// TIA Portal V17 export
// export: Created 2023-12-22T15:07:59.1760548Z, ExportSetting WithDefaults, DisplayName Totally Integrated Automation Portal, DisplayVersion V17, DisplayName TIA Portal Openness, DisplayVersion V17, DisplayName TIA Portal Version Control Interface, DisplayVersion V17, DisplayName STEP 7 Professional, DisplayVersion V17, DisplayName STEP 7 Safety, DisplayVersion V17, DisplayName WinCC Advanced, DisplayVersion V17
FUNCTION_BLOCK "PS_cnt"   // FB12, LAD
{ S7_Optimized_Access := 'FALSE' }
VERSION : 0.1
// stored: AutoNumber false, IsIECCheckEnabled false, SetENOAutomatically false, UDAEnableTagReadback false
   VAR_INPUT
      SP : Real;
      REQ : Int;
   END_VAR
   VAR_IN_OUT
      cnt : Int;   // Число насосов в работе
   END_VAR
   VAR DB_SPECIFIC
      Select_CMD : Bool;   // Запрос выбора насоса
      Select_Mode : Bool;   // 0 - для останова, 1 - для запуска
      Select_PS : Int;   // Выбранный насос
      PS_Add_Ready : Bool;   // Насосы вышли на общую точку
      PS_Add_CMD : Bool;   // Запрос выхода на общую точку
      SP_Low : Real := 40.0;   // Нижняя рабочая точка
      SP_High { S7_SetPoint := 'True'} : Real := 45.0;   // Верхняя рабочая точка
      SP_Min { S7_SetPoint := 'True'} : Real := 36.0;   // Точка открытия обратного клапана
      cnt_delta { S7_SetPoint := 'True'} : Real := 0.5;   // Смещение точки открытия обратного клапана на 1 работающий насос
      "Step" : Int;
      REQ_cnt : Int;
      PS_R_OFF : Int;   // Насос для отключения при ротации
      PS_R_ON : Int;   // Насос для запуска при ротации
      pos : Array[0..15] of Bool;
      tmp : Array[0..15] of Real;
   END_VAR
   VAR
      T_Delay_ON { S7_SetPoint := 'True'} : "Time_M";   // Задержка запуска след. насоса
      T_Delay_OFF { S7_SetPoint := 'True'} : "Time_M";   // Задержка останова след. насоса
   END_VAR
   VAR_TEMP
      x_delta : Real;
   END_VAR
   VAR_TEMP   // added for the SCL form of the ladder/FBD networks
      _w1 : Bool;
      _w2 : Bool;
      _w3 : Bool;
      _w4 : Bool;
      _w5 : Bool;
      _w6 : Bool;
      _w7 : Bool;
      _w8 : Bool;
   END_VAR
BEGIN

REGION Network 1: Коррекция нижней рабочей точки по числу насосов
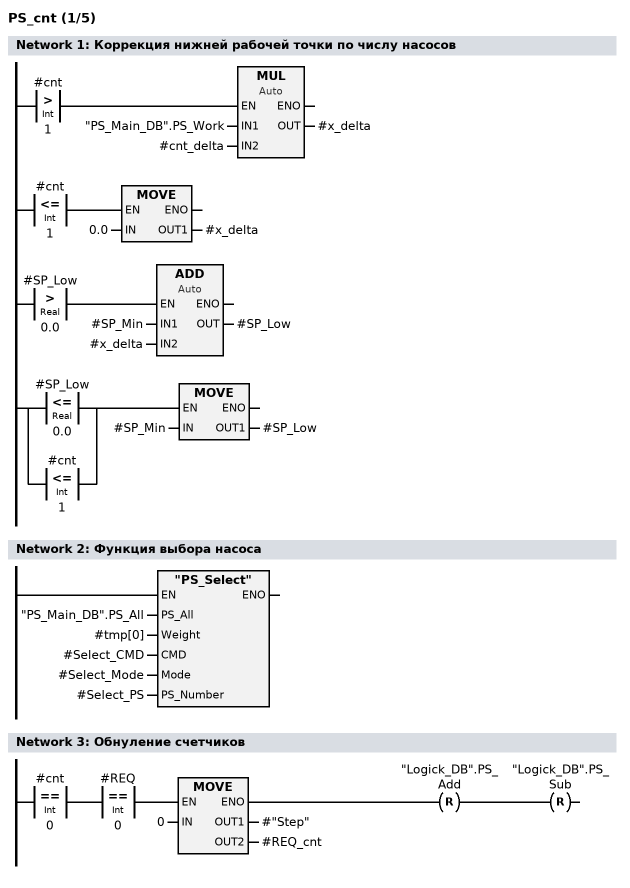
   RUNG wire#powerrail
      { S7_Templates := "SrcType := Int" } GT_Contact(in1 := #cnt, in2 := 1)
      Mul(in1 := "PS_Main_DB".PS_Work, in2 := #cnt_delta, out => #x_delta)
   END_RUNG
   RUNG wire#powerrail
      { S7_Templates := "SrcType := Int" } LE_Contact(in1 := #cnt, in2 := 1)
      Move(in := 0.0, out1 => #x_delta)
   END_RUNG
   RUNG wire#powerrail
      { S7_Templates := "SrcType := Real" } GT_Contact(in1 := #SP_Low, in2 := 0.0)
      Add(in1 := #SP_Min, in2 := #x_delta, out => #SP_Low)
   END_RUNG
   RUNG wire#powerrail
      { S7_Templates := "SrcType := Real" } LE_Contact(in1 := #SP_Low, in2 := 0.0)
      wire#w1
      Move(in := #SP_Min, out1 => #SP_Low)
   END_RUNG
   RUNG wire#powerrail
      { S7_Templates := "SrcType := Int" } LE_Contact(in1 := #cnt, in2 := 1)
   END_RUNG wire#w1
   // the same network as SCL:
   IF #cnt > 1 THEN #x_delta := "PS_Main_DB".PS_Work * #cnt_delta; END_IF;
   IF #cnt <= 1 THEN #x_delta := 0.0; END_IF;
   IF #SP_Low > 0.0 THEN #SP_Low := #SP_Min + #x_delta; END_IF;
   IF (#SP_Low <= 0.0) OR (#cnt <= 1) THEN #SP_Low := #SP_Min; END_IF;
END_REGION

REGION Network 2: Функция выбора насоса
   RUNG wire#powerrail
      "PS_Select"(PS_All := "PS_Main_DB".PS_All, Weight := #tmp[0], CMD := #Select_CMD, Mode := #Select_Mode, PS_Number := #Select_PS)
   END_RUNG
   // the same network as SCL:
   "PS_Select"(PS_All := "PS_Main_DB".PS_All,
               Weight := #tmp[0],
               CMD := #Select_CMD,
               Mode := #Select_Mode,
               PS_Number := #Select_PS);
END_REGION

REGION Network 3: Обнуление счетчиков
   RUNG wire#powerrail
      { S7_Templates := "SrcType := Int" } EQ_Contact(in1 := #cnt, in2 := 0)
      { S7_Templates := "SrcType := Int" } EQ_Contact(in1 := #REQ, in2 := 0)
      Move(in := 0, out1 => #"Step", out2 => #REQ_cnt)
      R_Coil( "Logick_DB".PS_Add )
      R_Coil( "Logick_DB".PS_Sub )
   END_RUNG
   // the same network as SCL:
   IF (#cnt = 0) AND (#REQ = 0) THEN
       #"Step" := 0;
       #REQ_cnt := 0;
       "Logick_DB".PS_Add := FALSE;
       "Logick_DB".PS_Sub := FALSE;
   END_IF;
END_REGION

REGION Network 4: Запуск первого насоса
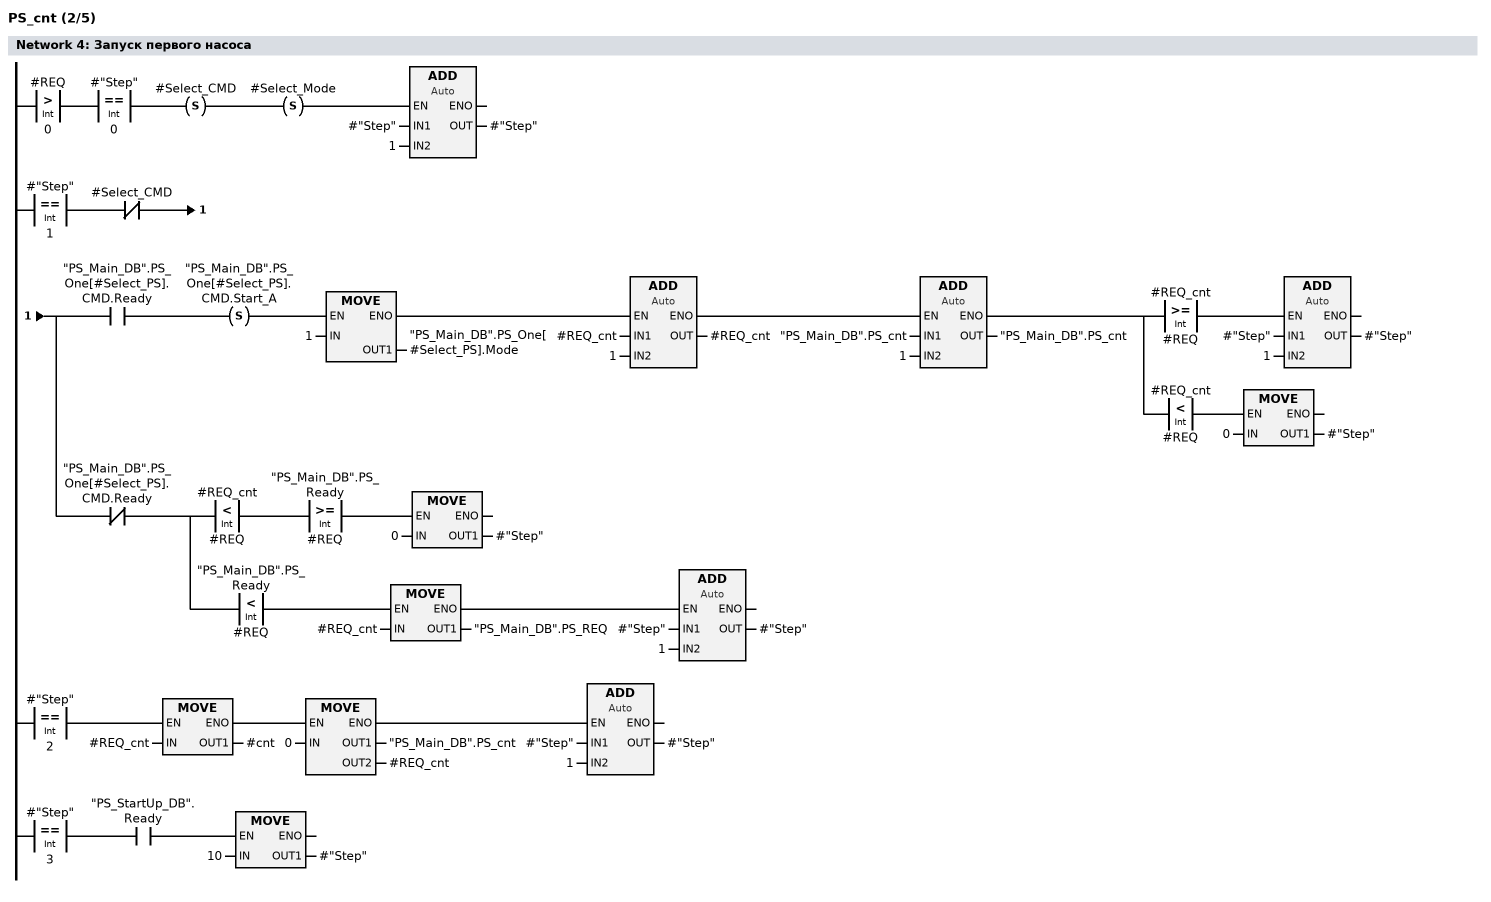
   RUNG wire#powerrail
      { S7_Templates := "SrcType := Int" } GT_Contact(in1 := #REQ, in2 := 0)
      { S7_Templates := "SrcType := Int" } EQ_Contact(in1 := #"Step", in2 := 0)
      S_Coil( #Select_CMD )
      S_Coil( #Select_Mode )
      Add(in1 := #"Step", in2 := 1, out => #"Step")
   END_RUNG
   RUNG wire#powerrail
      { S7_Templates := "SrcType := Int" } EQ_Contact(in1 := #"Step", in2 := 1)
      I_Contact( #Select_CMD )
      wire#w1
      Contact( "PS_Main_DB".PS_One[#Select_PS].CMD.Ready )
      S_Coil( "PS_Main_DB".PS_One[#Select_PS].CMD.Start_A )
      Move(in := 1, out1 => "PS_Main_DB".PS_One[#Select_PS].Mode)
      Add(in1 := #REQ_cnt, in2 := 1, out => #REQ_cnt)
      Add(in1 := "PS_Main_DB".PS_cnt, in2 := 1, out => "PS_Main_DB".PS_cnt)
      wire#w2
      { S7_Templates := "SrcType := Int" } GE_Contact(in1 := #REQ_cnt, in2 := #REQ)
      Add(in1 := #"Step", in2 := 1, out => #"Step")
   END_RUNG
   RUNG wire#w2
      { S7_Templates := "SrcType := Int" } LT_Contact(in1 := #REQ_cnt, in2 := #REQ)
      Move(in := 0, out1 => #"Step")
   END_RUNG
   RUNG wire#w1
      I_Contact( "PS_Main_DB".PS_One[#Select_PS].CMD.Ready )
      wire#w3
      { S7_Templates := "SrcType := Int" } LT_Contact(in1 := #REQ_cnt, in2 := #REQ)
      { S7_Templates := "SrcType := Int" } GE_Contact(in1 := "PS_Main_DB".PS_Ready, in2 := #REQ)
      Move(in := 0, out1 => #"Step")
   END_RUNG
   RUNG wire#w3
      { S7_Templates := "SrcType := Int" } LT_Contact(in1 := "PS_Main_DB".PS_Ready, in2 := #REQ)
      Move(in := #REQ_cnt, out1 => "PS_Main_DB".PS_REQ)
      Add(in1 := #"Step", in2 := 1, out => #"Step")
   END_RUNG
   RUNG wire#powerrail
      { S7_Templates := "SrcType := Int" } EQ_Contact(in1 := #"Step", in2 := 2)
      Move(in := #REQ_cnt, out1 => #cnt)
      Move(in := 0, out1 => "PS_Main_DB".PS_cnt, out2 => #REQ_cnt)
      Add(in1 := #"Step", in2 := 1, out => #"Step")
   END_RUNG
   RUNG wire#powerrail
      { S7_Templates := "SrcType := Int" } EQ_Contact(in1 := #"Step", in2 := 3)
      Contact( "PS_StartUp_DB".Ready )
      Move(in := 10, out1 => #"Step")
   END_RUNG
   // the same network as SCL:
   IF (#REQ > 0) AND (#"Step" = 0) THEN
       #Select_CMD := TRUE;
       #Select_Mode := TRUE;
       #"Step" := #"Step" + 1;
   END_IF;
   #_w1 := (#"Step" = 1) AND NOT #Select_CMD;
   #_w2 := #_w1 AND "PS_Main_DB".PS_One[#Select_PS].CMD.Ready;
   IF #_w2 THEN
       "PS_Main_DB".PS_One[#Select_PS].CMD.Start_A := TRUE;
       "PS_Main_DB".PS_One[#Select_PS].Mode := 1;
       #REQ_cnt := #REQ_cnt + 1;
       "PS_Main_DB".PS_cnt := "PS_Main_DB".PS_cnt + 1;
   END_IF;
   IF #_w2 AND (#REQ_cnt >= #REQ) THEN #"Step" := #"Step" + 1; END_IF;
   IF #_w2 AND (#REQ_cnt < #REQ) THEN #"Step" := 0; END_IF;
   #_w3 := #_w1 AND NOT "PS_Main_DB".PS_One[#Select_PS].CMD.Ready;
   IF #_w3 AND (#REQ_cnt < #REQ) AND ("PS_Main_DB".PS_Ready >= #REQ) THEN #"Step" := 0; END_IF;
   IF #_w3 AND ("PS_Main_DB".PS_Ready < #REQ) THEN
       "PS_Main_DB".PS_REQ := #REQ_cnt;
       #"Step" := #"Step" + 1;
   END_IF;
   IF #"Step" = 2 THEN
       #cnt := #REQ_cnt;
       "PS_Main_DB".PS_cnt := 0;
       #REQ_cnt := 0;
       #"Step" := #"Step" + 1;
   END_IF;
   IF (#"Step" = 3) AND "PS_StartUp_DB".Ready THEN #"Step" := 10; END_IF;
END_REGION

REGION Network 5: Добавление нового насоса
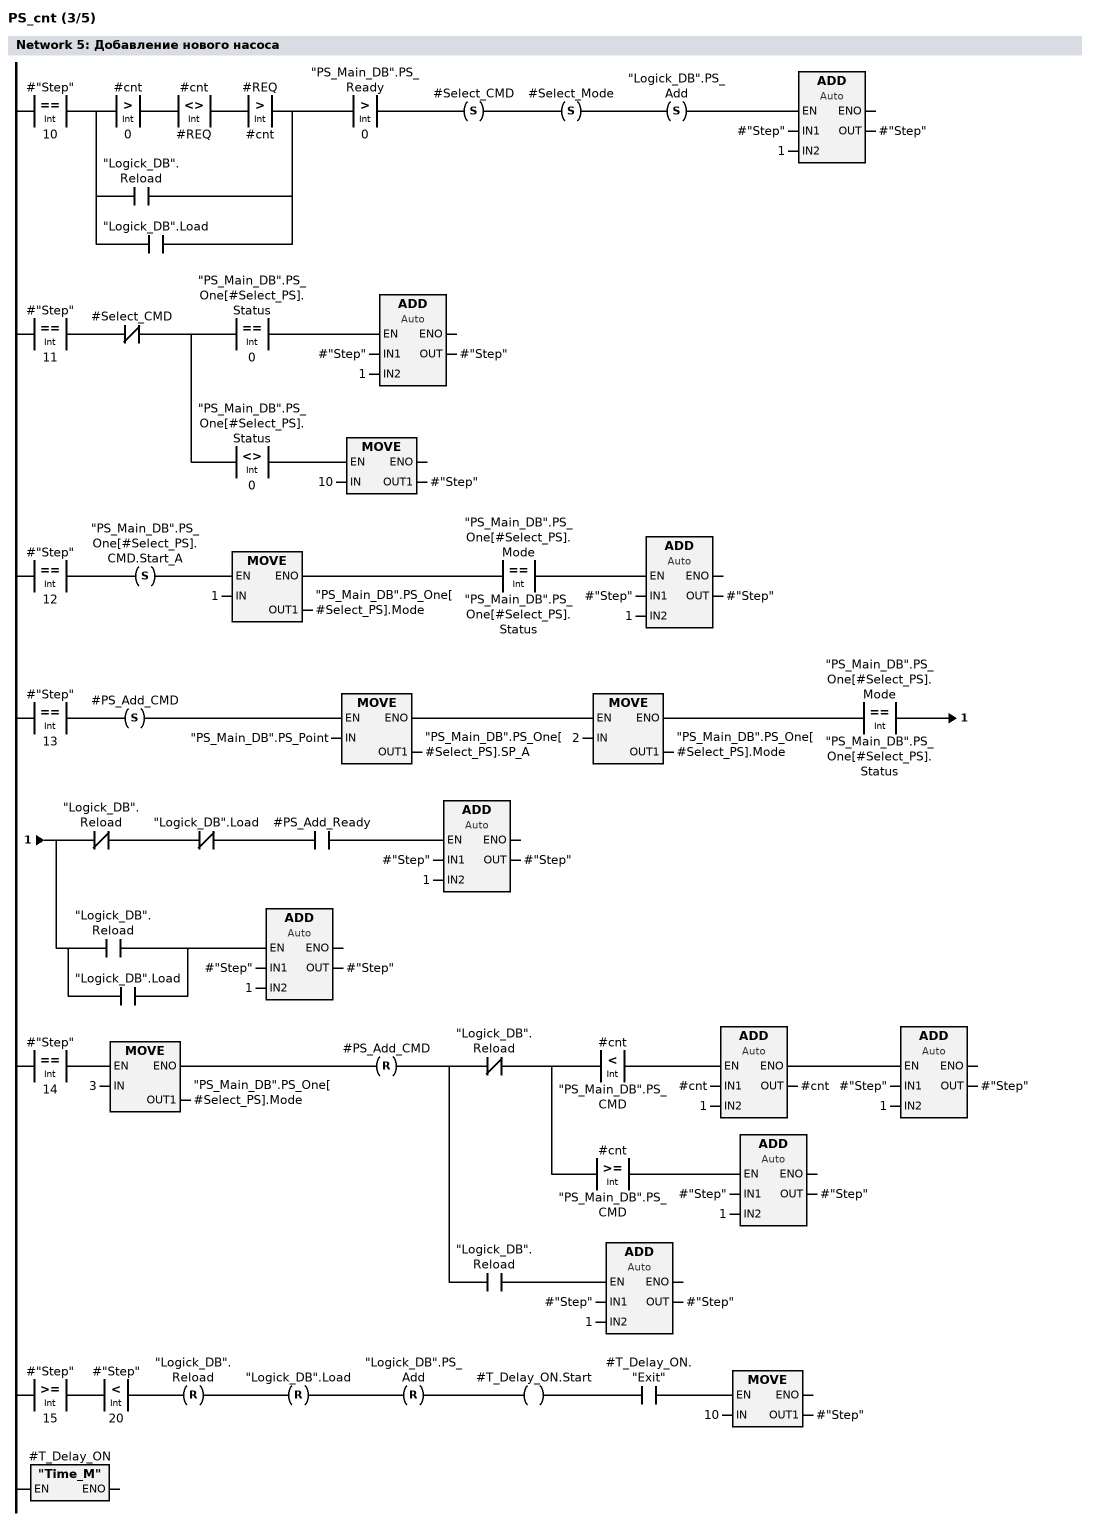
   RUNG wire#powerrail
      { S7_Templates := "SrcType := Int" } EQ_Contact(in1 := #"Step", in2 := 10)
      wire#w1
      { S7_Templates := "SrcType := Int" } GT_Contact(in1 := #cnt, in2 := 0)
      { S7_Templates := "SrcType := Int" } NE_Contact(in1 := #cnt, in2 := #REQ)
      { S7_Templates := "SrcType := Int" } GT_Contact(in1 := #REQ, in2 := #cnt)
      wire#w2
      { S7_Templates := "SrcType := Int" } GT_Contact(in1 := "PS_Main_DB".PS_Ready, in2 := 0)
      S_Coil( #Select_CMD )
      S_Coil( #Select_Mode )
      S_Coil( "Logick_DB".PS_Add )
      Add(in1 := #"Step", in2 := 1, out => #"Step")
   END_RUNG
   RUNG wire#w1
      Contact( "Logick_DB".Reload )
   END_RUNG wire#w2
   RUNG wire#w1
      Contact( "Logick_DB".Load )
   END_RUNG wire#w2
   RUNG wire#powerrail
      { S7_Templates := "SrcType := Int" } EQ_Contact(in1 := #"Step", in2 := 11)
      I_Contact( #Select_CMD )
      wire#w3
      { S7_Templates := "SrcType := Int" } EQ_Contact(in1 := "PS_Main_DB".PS_One[#Select_PS].Status, in2 := 0)
      Add(in1 := #"Step", in2 := 1, out => #"Step")
   END_RUNG
   RUNG wire#w3
      { S7_Templates := "SrcType := Int" } NE_Contact(in1 := "PS_Main_DB".PS_One[#Select_PS].Status, in2 := 0)
      Move(in := 10, out1 => #"Step")
   END_RUNG
   RUNG wire#powerrail
      { S7_Templates := "SrcType := Int" } EQ_Contact(in1 := #"Step", in2 := 12)
      S_Coil( "PS_Main_DB".PS_One[#Select_PS].CMD.Start_A )
      Move(in := 1, out1 => "PS_Main_DB".PS_One[#Select_PS].Mode)
      { S7_Templates := "SrcType := Int" } EQ_Contact(in1 := "PS_Main_DB".PS_One[#Select_PS].Mode, in2 := "PS_Main_DB".PS_One[#Select_PS].Status)
      Add(in1 := #"Step", in2 := 1, out => #"Step")
   END_RUNG
   RUNG wire#powerrail
      { S7_Templates := "SrcType := Int" } EQ_Contact(in1 := #"Step", in2 := 13)
      S_Coil( #PS_Add_CMD )
      Move(in := "PS_Main_DB".PS_Point, out1 => "PS_Main_DB".PS_One[#Select_PS].SP_A)
      Move(in := 2, out1 => "PS_Main_DB".PS_One[#Select_PS].Mode)
      { S7_Templates := "SrcType := Int" } EQ_Contact(in1 := "PS_Main_DB".PS_One[#Select_PS].Mode, in2 := "PS_Main_DB".PS_One[#Select_PS].Status)
      wire#w4
      I_Contact( "Logick_DB".Reload )
      I_Contact( "Logick_DB".Load )
      Contact( #PS_Add_Ready )
      Add(in1 := #"Step", in2 := 1, out => #"Step")
   END_RUNG
   RUNG wire#w4
      Contact( "Logick_DB".Reload )
      wire#w5
      Add(in1 := #"Step", in2 := 1, out => #"Step")
   END_RUNG
   RUNG wire#w4
      Contact( "Logick_DB".Load )
   END_RUNG wire#w5
   RUNG wire#powerrail
      { S7_Templates := "SrcType := Int" } EQ_Contact(in1 := #"Step", in2 := 14)
      Move(in := 3, out1 => "PS_Main_DB".PS_One[#Select_PS].Mode)
      R_Coil( #PS_Add_CMD )
      wire#w6
      I_Contact( "Logick_DB".Reload )
      wire#w7
      { S7_Templates := "SrcType := Int" } LT_Contact(in1 := #cnt, in2 := "PS_Main_DB".PS_CMD)
      Add(in1 := #cnt, in2 := 1, out => #cnt)
      Add(in1 := #"Step", in2 := 1, out => #"Step")
   END_RUNG
   RUNG wire#w7
      { S7_Templates := "SrcType := Int" } GE_Contact(in1 := #cnt, in2 := "PS_Main_DB".PS_CMD)
      Add(in1 := #"Step", in2 := 1, out => #"Step")
   END_RUNG
   RUNG wire#w6
      Contact( "Logick_DB".Reload )
      Add(in1 := #"Step", in2 := 1, out => #"Step")
   END_RUNG
   RUNG wire#powerrail
      { S7_Templates := "SrcType := Int" } GE_Contact(in1 := #"Step", in2 := 15)
      { S7_Templates := "SrcType := Int" } LT_Contact(in1 := #"Step", in2 := 20)
      R_Coil( "Logick_DB".Reload )
      R_Coil( "Logick_DB".Load )
      R_Coil( "Logick_DB".PS_Add )
      Coil( #T_Delay_ON.Start )
      Contact( #T_Delay_ON."Exit" )
      Move(in := 10, out1 => #"Step")
   END_RUNG
   RUNG wire#powerrail
      #T_Delay_ON()
   END_RUNG
   // the same network as SCL:
   IF (#"Step" = 10) AND (((#cnt > 0) AND (#cnt <> #REQ) AND (#REQ > #cnt)) OR "Logick_DB".Reload OR "Logick_DB".Load) AND ("PS_Main_DB".PS_Ready > 0) THEN
       #Select_CMD := TRUE;
       #Select_Mode := TRUE;
       "Logick_DB".PS_Add := TRUE;
       #"Step" := #"Step" + 1;
   END_IF;
   #_w1 := (#"Step" = 11) AND NOT #Select_CMD;
   IF #_w1 AND ("PS_Main_DB".PS_One[#Select_PS].Status = 0) THEN #"Step" := #"Step" + 1; END_IF;
   IF #_w1 AND ("PS_Main_DB".PS_One[#Select_PS].Status <> 0) THEN #"Step" := 10; END_IF;
   #_w2 := #"Step" = 12;
   IF #_w2 THEN
       "PS_Main_DB".PS_One[#Select_PS].CMD.Start_A := TRUE;
       "PS_Main_DB".PS_One[#Select_PS].Mode := 1;
   END_IF;
   IF #_w2 AND ("PS_Main_DB".PS_One[#Select_PS].Mode = "PS_Main_DB".PS_One[#Select_PS].Status) THEN
       #"Step" := #"Step" + 1;
   END_IF;
   #_w3 := #"Step" = 13;
   IF #_w3 THEN
       #PS_Add_CMD := TRUE;
       "PS_Main_DB".PS_One[#Select_PS].SP_A := "PS_Main_DB".PS_Point;
       "PS_Main_DB".PS_One[#Select_PS].Mode := 2;
   END_IF;
   #_w4 := #_w3 AND ("PS_Main_DB".PS_One[#Select_PS].Mode = "PS_Main_DB".PS_One[#Select_PS].Status);
   IF #_w4 AND NOT "Logick_DB".Reload AND NOT "Logick_DB".Load AND #PS_Add_Ready THEN
       #"Step" := #"Step" + 1;
   END_IF;
   IF #_w4 AND ("Logick_DB".Reload OR "Logick_DB".Load) THEN #"Step" := #"Step" + 1; END_IF;
   #_w5 := #"Step" = 14;
   IF #_w5 THEN
       "PS_Main_DB".PS_One[#Select_PS].Mode := 3;
       #PS_Add_CMD := FALSE;
   END_IF;
   #_w6 := #_w5 AND NOT "Logick_DB".Reload;
   #_w7 := #_w6 AND (#cnt < "PS_Main_DB".PS_CMD);
   IF #_w7 THEN
       #cnt := #cnt + 1;
       #"Step" := #"Step" + 1;
   END_IF;
   IF #_w6 AND (#cnt >= "PS_Main_DB".PS_CMD) THEN #"Step" := #"Step" + 1; END_IF;
   IF #_w5 AND "Logick_DB".Reload THEN #"Step" := #"Step" + 1; END_IF;
   #_w8 := (#"Step" >= 15) AND (#"Step" < 20);
   IF #_w8 THEN
       "Logick_DB".Reload := FALSE;
       "Logick_DB".Load := FALSE;
       "Logick_DB".PS_Add := FALSE;
   END_IF;
   #T_Delay_ON.Start := #_w8;
   IF #_w8 AND #T_Delay_ON."Exit" THEN #"Step" := 10; END_IF;
   #T_Delay_ON();   // "Time_M"
END_REGION

REGION Network 6: Вывод из работы насоса
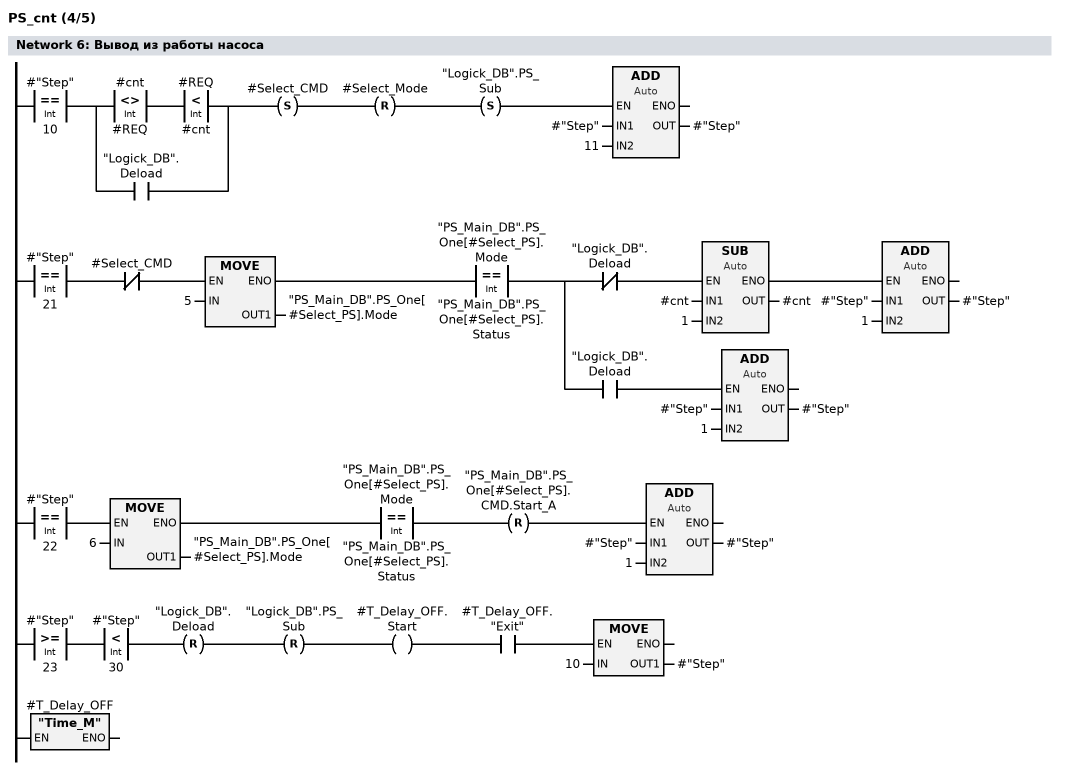
   RUNG wire#powerrail
      { S7_Templates := "SrcType := Int" } EQ_Contact(in1 := #"Step", in2 := 10)
      wire#w1
      { S7_Templates := "SrcType := Int" } NE_Contact(in1 := #cnt, in2 := #REQ)
      { S7_Templates := "SrcType := Int" } LT_Contact(in1 := #REQ, in2 := #cnt)
      wire#w2
      S_Coil( #Select_CMD )
      R_Coil( #Select_Mode )
      S_Coil( "Logick_DB".PS_Sub )
      Add(in1 := #"Step", in2 := 11, out => #"Step")
   END_RUNG
   RUNG wire#w1
      Contact( "Logick_DB".Deload )
   END_RUNG wire#w2
   RUNG wire#powerrail
      { S7_Templates := "SrcType := Int" } EQ_Contact(in1 := #"Step", in2 := 21)
      I_Contact( #Select_CMD )
      Move(in := 5, out1 => "PS_Main_DB".PS_One[#Select_PS].Mode)
      { S7_Templates := "SrcType := Int" } EQ_Contact(in1 := "PS_Main_DB".PS_One[#Select_PS].Mode, in2 := "PS_Main_DB".PS_One[#Select_PS].Status)
      wire#w3
      I_Contact( "Logick_DB".Deload )
      Sub(in1 := #cnt, in2 := 1, out => #cnt)
      Add(in1 := #"Step", in2 := 1, out => #"Step")
   END_RUNG
   RUNG wire#w3
      Contact( "Logick_DB".Deload )
      Add(in1 := #"Step", in2 := 1, out => #"Step")
   END_RUNG
   RUNG wire#powerrail
      { S7_Templates := "SrcType := Int" } EQ_Contact(in1 := #"Step", in2 := 22)
      Move(in := 6, out1 => "PS_Main_DB".PS_One[#Select_PS].Mode)
      { S7_Templates := "SrcType := Int" } EQ_Contact(in1 := "PS_Main_DB".PS_One[#Select_PS].Mode, in2 := "PS_Main_DB".PS_One[#Select_PS].Status)
      R_Coil( "PS_Main_DB".PS_One[#Select_PS].CMD.Start_A )
      Add(in1 := #"Step", in2 := 1, out => #"Step")
   END_RUNG
   RUNG wire#powerrail
      { S7_Templates := "SrcType := Int" } GE_Contact(in1 := #"Step", in2 := 23)
      { S7_Templates := "SrcType := Int" } LT_Contact(in1 := #"Step", in2 := 30)
      R_Coil( "Logick_DB".Deload )
      R_Coil( "Logick_DB".PS_Sub )
      Coil( #T_Delay_OFF.Start )
      Contact( #T_Delay_OFF."Exit" )
      Move(in := 10, out1 => #"Step")
   END_RUNG
   RUNG wire#powerrail
      #T_Delay_OFF()
   END_RUNG
   // the same network as SCL:
   IF (#"Step" = 10) AND (((#cnt <> #REQ) AND (#REQ < #cnt)) OR "Logick_DB".Deload) THEN
       #Select_CMD := TRUE;
       #Select_Mode := FALSE;
       "Logick_DB".PS_Sub := TRUE;
       #"Step" := #"Step" + 11;
   END_IF;
   #_w1 := (#"Step" = 21) AND NOT #Select_CMD;
   IF #_w1 THEN "PS_Main_DB".PS_One[#Select_PS].Mode := 5; END_IF;
   #_w2 := #_w1 AND ("PS_Main_DB".PS_One[#Select_PS].Mode = "PS_Main_DB".PS_One[#Select_PS].Status);
   IF #_w2 AND NOT "Logick_DB".Deload THEN
       #cnt := #cnt - 1;
       #"Step" := #"Step" + 1;
   END_IF;
   IF #_w2 AND "Logick_DB".Deload THEN #"Step" := #"Step" + 1; END_IF;
   #_w3 := #"Step" = 22;
   IF #_w3 THEN "PS_Main_DB".PS_One[#Select_PS].Mode := 6; END_IF;
   #_w4 := #_w3 AND ("PS_Main_DB".PS_One[#Select_PS].Mode = "PS_Main_DB".PS_One[#Select_PS].Status);
   IF #_w4 THEN
       "PS_Main_DB".PS_One[#Select_PS].CMD.Start_A := FALSE;
       #"Step" := #"Step" + 1;
   END_IF;
   #_w5 := (#"Step" >= 23) AND (#"Step" < 30);
   IF #_w5 THEN
       "Logick_DB".Deload := FALSE;
       "Logick_DB".PS_Sub := FALSE;
   END_IF;
   #T_Delay_OFF.Start := #_w5;
   IF #_w5 AND #T_Delay_OFF."Exit" THEN #"Step" := 10; END_IF;
   #T_Delay_OFF();   // "Time_M"
END_REGION

REGION Network 7: Ротация насосов
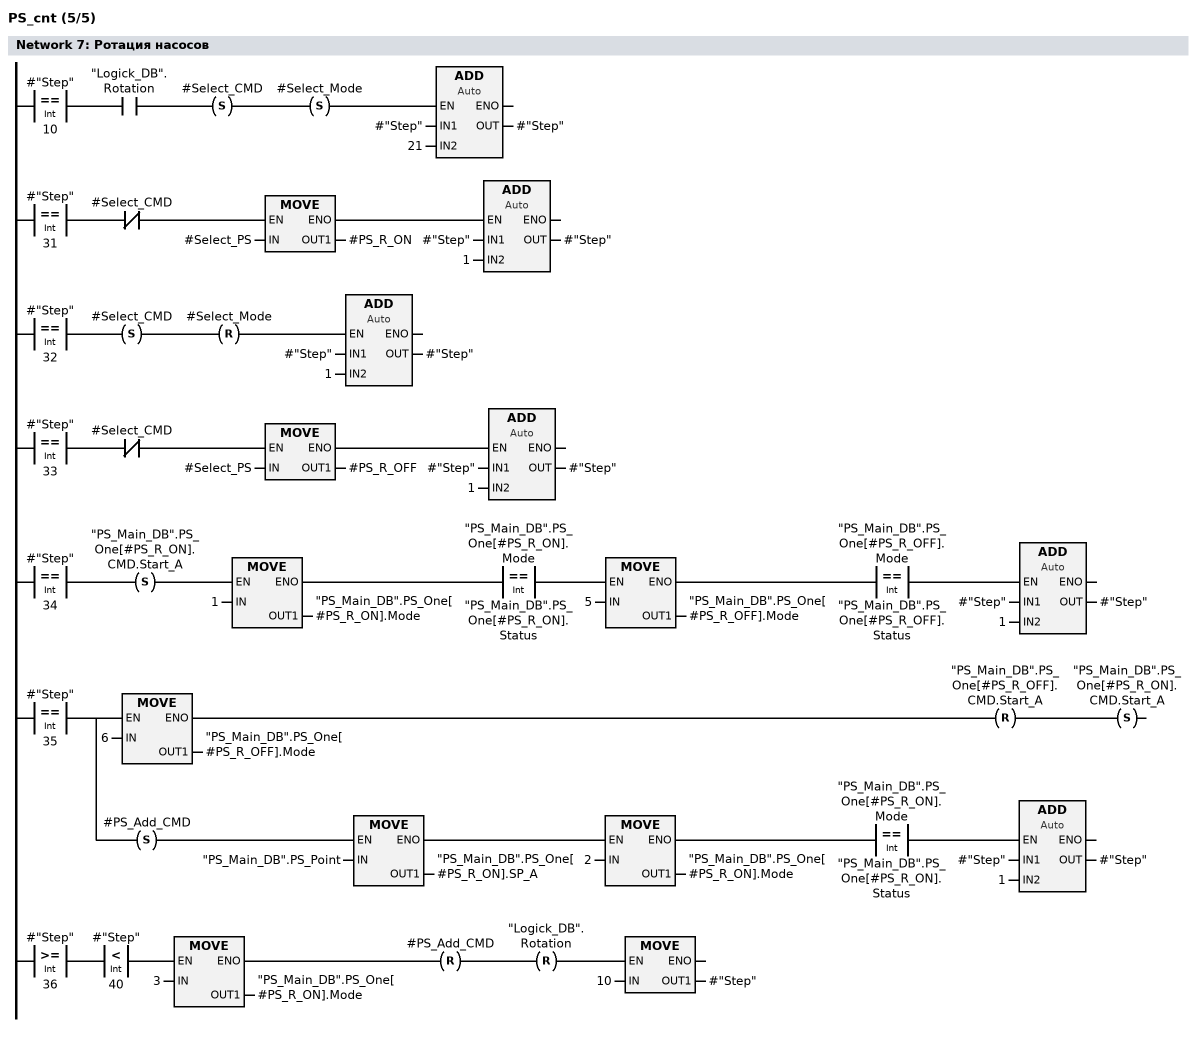
   RUNG wire#powerrail
      { S7_Templates := "SrcType := Int" } EQ_Contact(in1 := #"Step", in2 := 10)
      Contact( "Logick_DB".Rotation )
      S_Coil( #Select_CMD )
      S_Coil( #Select_Mode )
      Add(in1 := #"Step", in2 := 21, out => #"Step")
   END_RUNG
   RUNG wire#powerrail
      { S7_Templates := "SrcType := Int" } EQ_Contact(in1 := #"Step", in2 := 31)
      I_Contact( #Select_CMD )
      Move(in := #Select_PS, out1 => #PS_R_ON)
      Add(in1 := #"Step", in2 := 1, out => #"Step")
   END_RUNG
   RUNG wire#powerrail
      { S7_Templates := "SrcType := Int" } EQ_Contact(in1 := #"Step", in2 := 32)
      S_Coil( #Select_CMD )
      R_Coil( #Select_Mode )
      Add(in1 := #"Step", in2 := 1, out => #"Step")
   END_RUNG
   RUNG wire#powerrail
      { S7_Templates := "SrcType := Int" } EQ_Contact(in1 := #"Step", in2 := 33)
      I_Contact( #Select_CMD )
      Move(in := #Select_PS, out1 => #PS_R_OFF)
      Add(in1 := #"Step", in2 := 1, out => #"Step")
   END_RUNG
   RUNG wire#powerrail
      { S7_Templates := "SrcType := Int" } EQ_Contact(in1 := #"Step", in2 := 34)
      S_Coil( "PS_Main_DB".PS_One[#PS_R_ON].CMD.Start_A )
      Move(in := 1, out1 => "PS_Main_DB".PS_One[#PS_R_ON].Mode)
      { S7_Templates := "SrcType := Int" } EQ_Contact(in1 := "PS_Main_DB".PS_One[#PS_R_ON].Mode, in2 := "PS_Main_DB".PS_One[#PS_R_ON].Status)
      Move(in := 5, out1 => "PS_Main_DB".PS_One[#PS_R_OFF].Mode)
      { S7_Templates := "SrcType := Int" } EQ_Contact(in1 := "PS_Main_DB".PS_One[#PS_R_OFF].Mode, in2 := "PS_Main_DB".PS_One[#PS_R_OFF].Status)
      Add(in1 := #"Step", in2 := 1, out => #"Step")
   END_RUNG
   RUNG wire#powerrail
      { S7_Templates := "SrcType := Int" } EQ_Contact(in1 := #"Step", in2 := 35)
      wire#w1
      Move(in := 6, out1 => "PS_Main_DB".PS_One[#PS_R_OFF].Mode)
      R_Coil( "PS_Main_DB".PS_One[#PS_R_OFF].CMD.Start_A )
      S_Coil( "PS_Main_DB".PS_One[#PS_R_ON].CMD.Start_A )
   END_RUNG
   RUNG wire#w1
      S_Coil( #PS_Add_CMD )
      Move(in := "PS_Main_DB".PS_Point, out1 => "PS_Main_DB".PS_One[#PS_R_ON].SP_A)
      Move(in := 2, out1 => "PS_Main_DB".PS_One[#PS_R_ON].Mode)
      { S7_Templates := "SrcType := Int" } EQ_Contact(in1 := "PS_Main_DB".PS_One[#PS_R_ON].Mode, in2 := "PS_Main_DB".PS_One[#PS_R_ON].Status)
      Add(in1 := #"Step", in2 := 1, out => #"Step")
   END_RUNG
   RUNG wire#powerrail
      { S7_Templates := "SrcType := Int" } GE_Contact(in1 := #"Step", in2 := 36)
      { S7_Templates := "SrcType := Int" } LT_Contact(in1 := #"Step", in2 := 40)
      Move(in := 3, out1 => "PS_Main_DB".PS_One[#PS_R_ON].Mode)
      R_Coil( #PS_Add_CMD )
      R_Coil( "Logick_DB".Rotation )
      Move(in := 10, out1 => #"Step")
   END_RUNG
   // the same network as SCL:
   IF (#"Step" = 10) AND "Logick_DB".Rotation THEN
       #Select_CMD := TRUE;
       #Select_Mode := TRUE;
       #"Step" := #"Step" + 21;
   END_IF;
   IF (#"Step" = 31) AND NOT #Select_CMD THEN
       #PS_R_ON := #Select_PS;
       #"Step" := #"Step" + 1;
   END_IF;
   IF #"Step" = 32 THEN
       #Select_CMD := TRUE;
       #Select_Mode := FALSE;
       #"Step" := #"Step" + 1;
   END_IF;
   IF (#"Step" = 33) AND NOT #Select_CMD THEN
       #PS_R_OFF := #Select_PS;
       #"Step" := #"Step" + 1;
   END_IF;
   #_w1 := #"Step" = 34;
   IF #_w1 THEN
       "PS_Main_DB".PS_One[#PS_R_ON].CMD.Start_A := TRUE;
       "PS_Main_DB".PS_One[#PS_R_ON].Mode := 1;
   END_IF;
   #_w2 := #_w1 AND ("PS_Main_DB".PS_One[#PS_R_ON].Mode = "PS_Main_DB".PS_One[#PS_R_ON].Status);
   IF #_w2 THEN "PS_Main_DB".PS_One[#PS_R_OFF].Mode := 5; END_IF;
   IF #_w2 AND ("PS_Main_DB".PS_One[#PS_R_OFF].Mode = "PS_Main_DB".PS_One[#PS_R_OFF].Status) THEN
       #"Step" := #"Step" + 1;
   END_IF;
   #_w3 := #"Step" = 35;
   IF #_w3 THEN
       "PS_Main_DB".PS_One[#PS_R_OFF].Mode := 6;
       "PS_Main_DB".PS_One[#PS_R_OFF].CMD.Start_A := FALSE;
       "PS_Main_DB".PS_One[#PS_R_ON].CMD.Start_A := TRUE;
       #PS_Add_CMD := TRUE;
       "PS_Main_DB".PS_One[#PS_R_ON].SP_A := "PS_Main_DB".PS_Point;
       "PS_Main_DB".PS_One[#PS_R_ON].Mode := 2;
   END_IF;
   IF #_w3 AND ("PS_Main_DB".PS_One[#PS_R_ON].Mode = "PS_Main_DB".PS_One[#PS_R_ON].Status) THEN
       #"Step" := #"Step" + 1;
   END_IF;
   IF (#"Step" >= 36) AND (#"Step" < 40) THEN
       "PS_Main_DB".PS_One[#PS_R_ON].Mode := 3;
       #PS_Add_CMD := FALSE;
       "Logick_DB".Rotation := FALSE;
       #"Step" := 10;
   END_IF;
END_REGION
END_FUNCTION_BLOCK
